TYPE MyStructure :
STRUCT
	Name : STRING;
	Age : INT;
	Country : STRING;
END_STRUCT
END_TYPE

(* stored: Version 1.1.0.1, ProductVersion 3.1.4024.12
   DUT MyStructure: Id {07dcead1-0a38-4eea-91f7-f7ca26714027} *)
